// TIA Portal project "SCDW_Project" (V17)

(* hardware
DEVICE "PLC_1"  S7-1200 Station
   slot 0: "Rack_0"  S7-1200 Rack  Rack  V1.0
   slot 1: "PLC_1"  CPU 1214C AC/DC/Rly  6ES7 214-1BG40-0XB0  V4.5
   slot 2: "DI_16x24VDC_DQ_16xRelay_1"  6ES7 223-1PL30-0XB0  V1.0
   slot 101: "Module_101"  6ES7 241-1CH32-0XB0  V2.1
*)

// ===== PLC "PLC_1"  CPU 1214C AC/DC/Rly =====

VAR_GLOBAL   // PLC tag table "数字输入量模块3"
   "消音复位" AT %I6.2 : Bool;
   "燃气低压" AT %I6.3 : Bool;
   "燃气高压" AT %I6.4 : Bool;
   "燃气泄漏" AT %I6.5 : Bool;
   "急停" AT %I6.6 : Bool;
   "15#小火" AT %Q6.0 : Bool;
   "15#复位" AT %Q6.1 : Bool;
   "15#大火" AT %Q6.2 : Bool;
   "烧嘴电源" AT %Q6.5 : Bool;
   "蜂鸣器" AT %Q6.6 : Bool;
END_VAR

VAR_GLOBAL   // PLC tag table "数字输入量模块2"
   "11#小火反馈" AT %I4.0 : Bool;
   "11#故障反馈" AT %I4.1 : Bool;
   "11#大火反馈" AT %I4.2 : Bool;
   "12#小火反馈" AT %I4.3 : Bool;
   "12#故障反馈" AT %I4.4 : Bool;
   "12#大火反馈" AT %I4.5 : Bool;
   "13#小火反馈" AT %I4.6 : Bool;
   "13#故障反馈" AT %I4.7 : Bool;
   "13#大火反馈" AT %I5.0 : Bool;
   "14#小火反馈" AT %I5.1 : Bool;
   "14#故障反馈" AT %I5.2 : Bool;
   "14#大火反馈" AT %I5.3 : Bool;
   "15#小火反馈" AT %I5.4 : Bool;
   "15#故障反馈" AT %I5.5 : Bool;
   "15#大火反馈" AT %I5.6 : Bool;
   "9#大火" AT %Q4.0 : Bool;
   "10#小火" AT %Q4.1 : Bool;
   "10#复位" AT %Q4.2 : Bool;
   "10#大火" AT %Q4.3 : Bool;
   "11#小火" AT %Q4.4 : Bool;
   "11#复位" AT %Q4.5 : Bool;
   "11#大火" AT %Q4.6 : Bool;
   "12#小火" AT %Q4.7 : Bool;
   "12#复位" AT %Q5.0 : Bool;
   "12#大火" AT %Q5.1 : Bool;
   "13#小火" AT %Q5.2 : Bool;
   "13#复位" AT %Q5.3 : Bool;
   "13#大火" AT %Q5.4 : Bool;
   "14#小火" AT %Q5.5 : Bool;
   "14#复位" AT %Q5.6 : Bool;
   "14#大火" AT %Q5.7 : Bool;
END_VAR

VAR_GLOBAL   // PLC tag table "数字输入量模块1"
   "5#大火反馈" AT %I2.0 : Bool;
   "6#小火反馈" AT %I2.1 : Bool;
   "6#故障反馈" AT %I2.2 : Bool;
   "6#大火反馈" AT %I2.3 : Bool;
   "7#小火反馈" AT %I2.4 : Bool;
   "7#故障反馈" AT %I2.5 : Bool;
   "7#大火反馈" AT %I2.6 : Bool;
   "8#小火反馈" AT %I2.7 : Bool;
   "8#故障反馈" AT %I3.0 : Bool;
   "8#大火反馈" AT %I3.1 : Bool;
   "9#小火反馈" AT %I3.2 : Bool;
   "9#故障反馈" AT %I3.3 : Bool;
   "9#大火反馈" AT %I3.4 : Bool;
   "10#小火反馈" AT %I3.5 : Bool;
   "10#故障反馈" AT %I3.6 : Bool;
   "10#大火反馈" AT %I3.7 : Bool;
   "4#复位" AT %Q2.0 : Bool;
   "4#大火" AT %Q2.1 : Bool;
   "5#小火" AT %Q2.2 : Bool;
   "5#复位" AT %Q2.3 : Bool;
   "5#大火" AT %Q2.4 : Bool;
   "6#小火" AT %Q2.5 : Bool;
   "6#复位" AT %Q2.6 : Bool;
   "6#大火" AT %Q2.7 : Bool;
   "7#小火" AT %Q3.0 : Bool;
   "7#复位" AT %Q3.1 : Bool;
   "7#大火" AT %Q3.2 : Bool;
   "8#小火" AT %Q3.3 : Bool;
   "8#复位" AT %Q3.4 : Bool;
   "8#大火" AT %Q3.5 : Bool;
   "9#小火" AT %Q3.6 : Bool;
   "9#复位" AT %Q3.7 : Bool;
END_VAR

VAR_GLOBAL   // PLC tag table "cpu点表"
   "1#小火反馈" AT %I0.0 : Bool;
   "1#故障反馈" AT %I0.1 : Bool;
   "1#大火反馈" AT %I0.2 : Bool;
   "2#小火反馈" AT %I0.3 : Bool;
   "2#故障反馈" AT %I0.4 : Bool;
   "2#大火反馈" AT %I0.5 : Bool;
   "3#小火反馈" AT %I0.6 : Bool;
   "3#故障反馈" AT %I0.7 : Bool;
   "3#大火反馈" AT %I1.0 : Bool;
   "4#小火反馈" AT %I1.1 : Bool;
   "4#故障反馈" AT %I1.2 : Bool;
   "4#大火反馈" AT %I1.3 : Bool;
   "5#小火反馈" AT %I1.4 : Bool;
   "5#故障反馈" AT %I1.5 : Bool;
   "1#小火" AT %Q0.0 : Bool;
   "1#复位" AT %Q0.1 : Bool;
   "1#大火" AT %Q0.2 : Bool;
   "2#小火" AT %Q0.3 : Bool;
   "2#复位" AT %Q0.4 : Bool;
   "2#大火" AT %Q0.5 : Bool;
   "3#小火" AT %Q0.6 : Bool;
   "3#复位" AT %Q0.7 : Bool;
   "3#大火" AT %Q1.0 : Bool;
   "4#小火" AT %Q1.1 : Bool;
   "风压" AT %IW64 : Int;
END_VAR

DATA_BLOCK "风机DB"   // DB1
{ S7_Optimized_Access := 'TRUE' }
VERSION : 0.1
   VAR
      风机运行按钮 : Bool;
      风机故障反馈 : Bool;
      风机运行标志 : Bool;
      风机运行反馈 : Bool;
      风机复位标志 : Bool;
      风机手动 : Bool;
      PID控制 : Bool;
      风压故障 : Bool;
      运行数据组_1 : Bool;   // 运行数据组[1]
      运行数据组_8 : Bool;   // 运行数据组[8]
      反馈数据组_0 : Bool;   // 反馈数据组[0]
      反馈数据组_12 : Bool;   // 反馈数据组[12]
      变频器通讯运行状态 : Int;
      变频器通讯反馈频率 : Int;
      变频器通讯设定运行 : Int;
      变频器通讯设定频率 : Int;
      风机过渡 : Int;
      风压转换过渡 : Real;
      风机转换过渡 : Real;
      风机控制输出码值 : Real;
      风机手动频率 : Real;
      风机自动输出 : Real;
      风机控制输出 : Real;
      风机反馈频率 : Real;
      _1_8区通讯延时定时器 : IEC_TIMER;
      _9_15区通讯延时定时器 : IEC_TIMER;
      变频器通讯延时定时器 : IEC_TIMER;
   END_VAR
BEGIN
END_DATA_BLOCK

FUNCTION "风机输出功能" : Void   // FC1, LAD
{ S7_Optimized_Access := 'TRUE' }
VERSION : 0.1
BEGIN

REGION Network 1
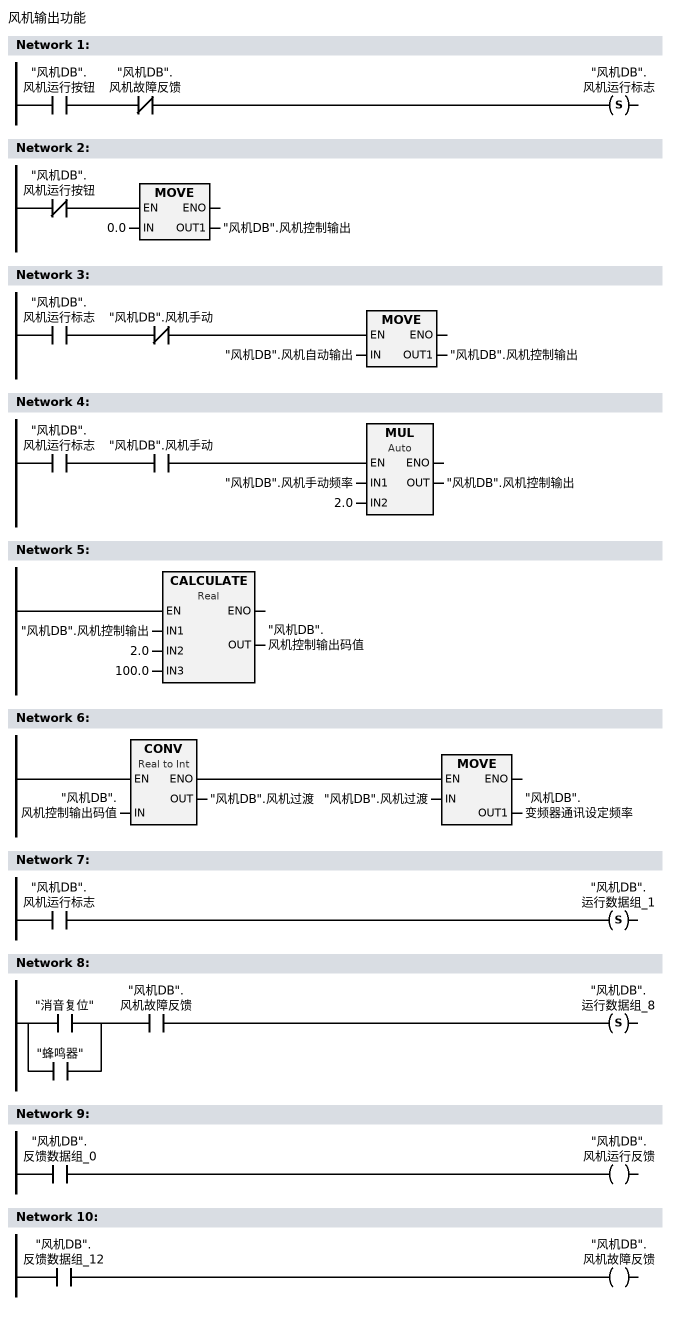
   RUNG wire#powerrail
      Contact( "风机DB".风机运行按钮 )
      I_Contact( "风机DB".风机故障反馈 )
      S_Coil( "风机DB".风机运行标志 )
   END_RUNG
   // the same network as SCL:
   IF "风机DB".风机运行按钮 AND NOT "风机DB".风机故障反馈 THEN "风机DB".风机运行标志 := TRUE; END_IF;
END_REGION

REGION Network 2
   RUNG wire#powerrail
      I_Contact( "风机DB".风机运行按钮 )
      { S7_GenerateENO := "TRUE" } Move(in := 0.0, out1 => "风机DB".风机控制输出)
   END_RUNG
   // the same network as SCL:
   IF NOT "风机DB".风机运行按钮 THEN "风机DB".风机控制输出 := 0.0; END_IF;
END_REGION

REGION Network 3
   RUNG wire#powerrail
      Contact( "风机DB".风机运行标志 )
      I_Contact( "风机DB".风机手动 )
      { S7_GenerateENO := "TRUE" } Move(in := "风机DB".风机自动输出, out1 => "风机DB".风机控制输出)
   END_RUNG
   // the same network as SCL:
   IF "风机DB".风机运行标志 AND NOT "风机DB".风机手动 THEN "风机DB".风机控制输出 := "风机DB".风机自动输出; END_IF;
END_REGION

REGION Network 4
   RUNG wire#powerrail
      Contact( "风机DB".风机运行标志 )
      Contact( "风机DB".风机手动 )
      { S7_GenerateENO := "TRUE" } Mul(in1 := "风机DB".风机手动频率, in2 := 2.0, out => "风机DB".风机控制输出)
   END_RUNG
   // the same network as SCL:
   IF "风机DB".风机运行标志 AND "风机DB".风机手动 THEN "风机DB".风机控制输出 := "风机DB".风机手动频率 * 2.0; END_IF;
END_REGION

REGION Network 5
   RUNG wire#powerrail
      { S7_Templates := "SrcType := Real"; S7_GenerateENO := "TRUE"; S7_Expression := "(IN1/IN2)*IN3" } Calculate(in1 := "风机DB".风机控制输出, in2 := 2.0, in3 := 100.0, out => "风机DB".风机控制输出码值)
   END_RUNG
   // the same network as SCL:
   "风机DB".风机控制输出码值 := ("风机DB".风机控制输出/2.0)*100.0;
END_REGION

REGION Network 6
   RUNG wire#powerrail
      { S7_Templates := "[SrcType := Real, DestType := Int]"; S7_GenerateENO := "TRUE" } Convert(in := "风机DB".风机控制输出码值, out => "风机DB".风机过渡)
      { S7_GenerateENO := "TRUE" } Move(in := "风机DB".风机过渡, out1 => "风机DB".变频器通讯设定频率)
   END_RUNG
   // the same network as SCL:
   // ENO of a box is taken as its EN; it also drops when the box reports an error
   "风机DB".风机过渡 := REAL_TO_INT("风机DB".风机控制输出码值);
   "风机DB".变频器通讯设定频率 := "风机DB".风机过渡;
END_REGION

REGION Network 7
   RUNG wire#powerrail
      Contact( "风机DB".风机运行标志 )
      S_Coil( "风机DB".运行数据组_1 )
   END_RUNG
   // the same network as SCL:
   IF "风机DB".风机运行标志 THEN "风机DB".运行数据组_1 := TRUE; END_IF;
END_REGION

REGION Network 8
   RUNG wire#powerrail
      Contact( "消音复位" )
      wire#w1
      Contact( "风机DB".风机故障反馈 )
      S_Coil( "风机DB".运行数据组_8 )
   END_RUNG
   RUNG wire#powerrail
      Contact( "蜂鸣器" )
   END_RUNG wire#w1
   // the same network as SCL:
   IF ("消音复位" OR "蜂鸣器") AND "风机DB".风机故障反馈 THEN "风机DB".运行数据组_8 := TRUE; END_IF;
END_REGION

REGION Network 9
   RUNG wire#powerrail
      Contact( "风机DB".反馈数据组_0 )
      Coil( "风机DB".风机运行反馈 )
   END_RUNG
   // the same network as SCL:
   "风机DB".风机运行反馈 := "风机DB".反馈数据组_0;
END_REGION

REGION Network 10
   RUNG wire#powerrail
      Contact( "风机DB".反馈数据组_12 )
      Coil( "风机DB".风机故障反馈 )
   END_RUNG
   // the same network as SCL:
   "风机DB".风机故障反馈 := "风机DB".反馈数据组_12;
END_REGION
END_FUNCTION

ORGANIZATION_BLOCK "Main"   // OB1, LAD, ProgramCycle
TITLE = "Main Program Sweep (Cycle)"
{ S7_Optimized_Access := 'TRUE' }
VERSION : 0.1
   VAR_INPUT
      Initial_Call : Bool;   // Initial call of this OB
      Remanence : Bool;   // =True, if remanent data are available
   END_VAR
BEGIN
END_ORGANIZATION_BLOCK